TYPE ST_RegistroDeTiempoEmpleado :
STRUCT
	stEmpleado : ST_Empleado; // Datos de la función Empleado
    stHorario  : ST_Horario;
END_STRUCT
END_TYPE

(* stored: Version 1.1.0.1, ProductVersion 3.1.4024.12
   DUT ST_RegistroDeTiempoEmpleado: Id {9f446250-ab40-4559-9646-3742b9b855d1} *)
